(* IEC 61131-3 sources: lasal-git-demo/CPU/LasalDemoProject/Class/DemoClass, 1 file *)

(* ---- DemoClass.st ---- *)
(*!
<Class
	Name               = "DemoClass"
	Revision           = "0.0"
	RealtimeTask       = "false"
	CyclicTask         = "true"
	DefCyclictime      = "1 ms"
	BackgroundTask     = "false"
	Sigmatek           = "false"
	OSInterface        = "false"
	HighPriority       = "false"
	Automatic          = "false"
	UpdateMode         = "Prescan"
	SharedCommandTable = "true"
	Objectsize         = "(422,120)">
	<Channels>
		<Server Name="ClassSvr" Visualized="false" Initialize="false" WriteProtected="true" Retentive="false"/>
		<Server
			Name           = "sDemoServer"
			Visualized     = "false"
			Initialize     = "false"
			WriteProtected = "false"
			Retentive      = "File">
			<OPCSettingsDefault Visible="true" WriteProtected="false"/>
		</Server>
		<Client Name="cDemoClient" Required="true" Internal="false"/>
	</Channels>
</Class>
*)
DemoClass : CLASS
  //Servers:
	ClassSvr 	: SvrChCmd_DINT;
	sDemoServer 	: SvrCh_DINT;
  //Clients:
	cDemoClient 	: CltCh_DINT;
  //Variables:
		vDemoVariable 	: DINT;
  //Functions:

	FUNCTION VIRTUAL GLOBAL CyWork
		VAR_INPUT
			EAX 	: UDINT;
		END_VAR
		VAR_OUTPUT
			state (EAX) 	: UDINT;
		END_VAR;
  //Tables:
	FUNCTION @STD
		VAR_OUTPUT
			ret_code	: CONFSTATES;
		END_VAR;
	FUNCTION GLOBAL TAB @CT_;
END_CLASS;

FUNCTION VIRTUAL GLOBAL DemoClass::CyWork
	VAR_INPUT
		EAX 	: UDINT;
	END_VAR
	VAR_OUTPUT
		state (EAX) 	: UDINT;
	END_VAR

	state := READY;

END_FUNCTION
